# EPICS substitutions: hytec8413TestApp/Db/ip231.substitutions
#==============================================================================
#
# Abs:  Acromag IP-231 DAC template
#
# Name: ip231.substitutions
#
#  Auth: 10-Aug-2006, S. Peng         (PENG)
#  Rev:  dd-mmm-yyyy, Reviewer's Name (USERNAME)
#-----------------------------------------------------------------------------
# Mod:
#       05-Dec-2007, K. Luchini       (LUCHINI):
#          changed record name substitutions
#
#==============================================================================
#
file IP231.template
{
  pattern { RECNAME              , CARD  ,  CH, EFUG,  EGUL , ADEL,  MDEL, HIHI,  HIGH, LOW, LOLO, EGU   }
          { "DAC:IN20:101:VSETPT", "ao0" ,   0, 10.0,  -10.0, 0.0 ,  0.0 , 4.5 ,  4.0 , 1.0, 0.5,  Volts }
          { "DAC:IN20:102:VSETPT", "ao0" ,   1, 10.0,  -10.0, 0.0 ,  0.0 , 4.5 ,  4.0 , 1.0, 0.5,  Volts }
          { "DAC:IN20:103:VSETPT", "ao0" ,   2, 10.0,  -10.0, 0.0 ,  0.0 , 4.5 ,  4.0 , 1.0, 0.5,  Volts }
          { "DAC:IN20:104:VSETPT", "ao0" ,   3, 10.0,  -10.0, 0.0 ,  0.0 , 4.5 ,  4.0 , 1.0, 0.5,  Volts }
          { "DAC:IN20:105:VSETPT", "ao0" ,   4, 10.0,  -10.0, 0.0 ,  0.0 , 4.5 ,  4.0 , 1.0, 0.5,  Volts }
          { "DAC:IN20:106:VSETPT", "ao0" ,   5, 10.0,  -10.0, 0.0 ,  0.0 , 4.5 ,  4.0 , 1.0, 0.5,  Volts }
          { "DAC:IN20:107:VSETPT", "ao0" ,   6, 10.0,  -10.0, 0.0 ,  0.0 , 4.5 ,  4.0 , 1.0, 0.5,  Volts }
          { "DAC:IN20:108:VSETPT", "ao0" ,   7, 10.0,  -10.0, 0.0 ,  0.0 , 4.5 ,  4.0 , 1.0, 0.5,  Volts }
          { "DAC:IN20:109:VSETPT", "ao0" ,   8, 10.0,  -10.0, 0.0 ,  0.0 , 4.5 ,  4.0 , 1.0, 0.5,  Volts }
          { "DAC:IN20:110:VSETPT", "ao0" ,   9, 10.0,  -10.0, 0.0 ,  0.0 , 4.5 ,  4.0 , 1.0, 0.5,  Volts }
          { "DAC:IN20:111:VSETPT", "ao0" ,  10, 10.0,  -10.0, 0.0 ,  0.0 , 4.5 ,  4.0 , 1.0, 0.5,  Volts }
          { "DAC:IN20:112:VSETPT", "ao0" ,  11, 10.0,  -10.0, 0.0 ,  0.0 , 4.5 ,  4.0 , 1.0, 0.5,  Volts }
          { "DAC:IN20:113:VSETPT", "ao0" ,  12, 10.0,  -10.0, 0.0 ,  0.0 , 4.5 ,  4.0 , 1.0, 0.5,  Volts }
          { "DAC:IN20:114:VSETPT", "ao0" ,  13, 10.0,  -10.0, 0.0 ,  0.0 , 4.5 ,  4.0 , 1.0, 0.5,  Volts }
          { "DAC:IN20:115:VSETPT", "ao0" ,  14, 10.0,  -10.0, 0.0 ,  0.0 , 4.5 ,  4.0 , 1.0, 0.5,  Volts }
          { "DAC:IN20:116:VSETPT", "ao0" ,  15, 10.0,  -10.0, 0.0 ,  0.0 , 4.5 ,  4.0 , 1.0, 0.5,  Volts }
}
